FUNCTION_BLOCK Pneumatics (* Composite Function Block Type *)
  (* Standard: 61499-2 *)
  (* Version 0.0, 2/14/2021, prana, nxtControl GmbH, template *)
  PACKAGE Main;
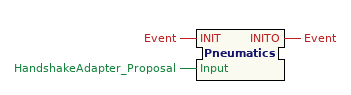
  EVENT_INPUT
    INIT; (* Initialization Request *)
  END_EVENT
  EVENT_OUTPUT
    INITO; (* Initialization Confirm *)
  END_EVENT
  SOCKETS
    Input : HandshakeAdapter_Proposal;
  END_SOCKETS
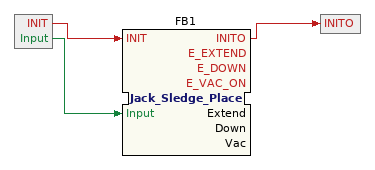
  FBS
    FB1 : Jack_Sledge_Place;
  END_FBS
  EVENT_CONNECTIONS
    INIT TO FB1.INIT;
    FB1.INITO TO INITO;
  END_CONNECTIONS
  ADAPTER_CONNECTIONS
    Input TO FB1.Input;
  END_CONNECTIONS
END_FUNCTION_BLOCK
